FUNCTION_BLOCK FB_TemperaturePIDControl
VAR_INPUT
END_VAR
VAR_OUTPUT
END_VAR
VAR
	rInput: REAL;
	// PID parameters
	rIprior: REAL := 0;
	rIterationtime: REAL := 6;
	reprior: REAL := 0;
	rPB: REAL :=9;
	rTi: REAL := 300;
	rTd: REAL := 90;
	rKp: REAL := 100/rPB;
	rKi: REAL := 1/rTi;
	rKd: REAL := 1/rTd;
	rBias: REAL := 0;
	// IO, HMI variables
	ryT: REAL; // Temperature measurement
	rspT: REAL; // Temperature setpoint
	buT: BOOL; // Temperature control (contactor)
	bTempCon: BOOL; // Temperature control mode (AUTO == 1, MAN == 0)
	//
	rontime: REAL;
	re: REAL;
	rI: REAL;
	// Cycle timer
	bCycleTimerStart : BOOL := 0;
	fbCycleTimer : TON; // EHKÄ TÄHÄN mielummin IN parametri kuin pT? uusi pt sitten koodissa aina? tai sitten kaikki inputit ja outputit tähän?
	// Ctrl timer
	bCtrlTimerStart : BOOL := 0;
	fbCtrlTimer : TON;	
	//
	rPIDypercentage: REAL;
	bAutomode: BOOL;
	bPercentageMode: BOOL;
END_VAR

IF ReactorTemperatureControl.iCycleTime <> 0 THEN
	rIterationTime := ReactorTemperatureControl.iCycleTime;
END_IF
IF ReactorTemperatureControl.iProportionalBand <> 0 THEN
	rPB := ReactorTemperatureControl.iProportionalBand;
END_IF
IF ReactorTemperatureControl.iIntegralTime <> 0 THEN
	rTi := ReactorTemperatureControl.iIntegralTime;
END_IF
IF ReactorTemperatureControl.iDerivativeTime <> 0 THEN
	rTd := ReactorTemperatureControl.iDerivativeTime;
END_IF
IF ReactorTemperatureControl.iBias <> 0 THEN
	rBias := ReactorTemperatureControl.iBias;
END_IF
//IO.bOutput := HMI.bContactor;
ReactorTemperatureControl.iTemperatureDisplayValue := GVL_IO.reactorTemperatureUpper/10;
//Temperature Control state
IF ReactorTemperatureControl.bTemperatureControlSwitch = 1 THEN
	ReactorTemperatureControl.sTemperatureControlState := 'AUTO';
END_IF
IF ReactorTemperatureControl.bTemperatureControlSwitch = 0 THEN
	ReactorTemperatureControl.sTemperatureControlState := 'MAN';
END_IF
// Read measurement values
// Temperature
ryT := INT_TO_FLOAT(in := GVL_IO.reactorTemperatureUpper);
ryT := ryT/10;
rspT := ReactorTemperatureControl.iTemperatureSetpoint;
buT := GVL_IO.reactorTemperatureContactor;
bTempCon := ReactorTemperatureControl.bTemperatureControlSwitch;
// Temperature PID control
fbCtrlTimer(IN := bCtrlTimerStart,PT := REAL_TO_TIME(rontime*1000));
fbCycleTimer(IN := bCycleTimerStart,PT := REAL_TO_TIME(rIterationtime*1000));
IF bTempCon = 1 THEN
	ReactorTemperatureControl.iTemperatureControlPercentage := 0;
	IF bCycleTimerStart = 0 THEN
		F_GetPIDOntime(rspT := rspT, ryT := ryT, rIprior := rIprior, riterationtime := riterationtime, reprior := reprior, rKp := rKp, rKi := rKi, rKd := rKd, rbias := rbias, rontime =>rontime, re => re, rI => rI);
		reprior := re;
		rIprior := rI;
		bCycleTimerStart := 1;
		bCtrlTimerStart := 1;
	ELSE
		F_ContactorControl(bCtrltimerQ := fbCtrlTimer.Q);
		IF fbCycleTimer.Q = 1 THEN
			bCycleTimerStart := 0;
			bCtrlTimerStart := 0;	
		END_IF
	END_IF
	bAutomode := 1;
	bPercentageMode := 0;
ELSE
	IF bAutomode THEN
		GVL_IO.reactorTemperatureContactor := 0;
		bAutomode := 0;
	END_IF
	rPIDypercentage := INT_TO_REAL(ReactorTemperatureControl.iTemperatureControlPercentage)/100;
	IF rPIDypercentage > 0 THEN
		bPercentageMode := TRUE;
		rontime := F_PercentageToTime(rPIDypercentage := rPIDypercentage,rIterationtime := rIterationtime);
		IF FbCycleTimer.Q = 0 THEN
			bCycleTimerStart := 1;
			bCtrlTimerStart := 1;
			F_ContactorControl(bCtrltimerQ := fbCtrlTimer.Q);
		END_IF
			IF fbCycleTimer.Q = 1 THEN
				bCycleTimerStart := 0;
				bCtrlTimerStart := 0;	
			END_IF	
	ELSIF rPIDypercentage = 0 THEN
		IF GVL_IO.reactorTemperatureContactor = 1 AND bPercentageMode THEN
			GVL_IO.reactorTemperatureContactor := 0;
		END_IF
		bPercentageMode := FALSE;
	END_IF
END_IF

END_FUNCTION_BLOCK

(* stored: Version 1.1.0.1, ProductVersion 3.1.4024.9
   POU FB_TemperaturePIDControl: Id {fec9367a-41a1-444a-b23a-817c84e06e42}, SpecialFunc None *)
